VAR_GLOBAL
    // Achsen ***************************************************	
	X_Achse_steuern						: DUT_Achse_Steuern;	
	X_Achse_status						: DUT_Achse_Status;	
		                            	
	Y_Achse_steuern						: DUT_Achse_Steuern;		
	Y_Achse_status						: DUT_Achse_Status;		

    // Frequenzumrichter ****************************************
	Bohraggr_Schluessel_ob_steuern		: DUT_SEW_FU_Steuern;	
	Bohraggr_Schluessel_ob_status		: DUT_SEW_FU_Status;

    // Ventile **************************************************
    Schluessel_ob_Bohrhub          		: DUT_Ventil_sps;

    // interne Variablen ****************************************
    sk_Freigabe                         : BOOL;
    sk                                  : INT;
    transport_einfoerdern_bereit        : BOOL;
    transport_ausfoerdern_bereit        : BOOL;

    Tuer_Anwahl                         : BOOL;   // Signal Tür Anwahl, Tür soll geöffnet werden
    Tuer_Freigabe                       : BOOL;   // Signal Tür Freigabe, Tür kann geöffnet werden
	
    // NCI Variablen *********************************************
	NCI_Steuern						: DUT_NCI_Steuern;
	NCI_Status						: DUT_NCI_Status;
	NCI_RPara_anNC					: ARRAY [0..99] OF LREAL;
	NCI_RPara_vonNC					: ARRAY [0..99] OF LREAL;
END_VAR

(* stored: Version 1.1.0.1
   GVL GVL_3400: Id {0c704e64-794b-4d8d-97d7-176fc5bac295} *)
